# EPICS substitutions: blenApp/Db/common/IMAXScale.substitutions
#==============================================================================
#
# Abs:  IMAX scale substitutions file.
#
# Name: IMAXScale.substitutions
#
# Note: Must follow the LCLS naming conventions.
#
#==============================================================================
#
file IMAXScaleCalc.db
{
pattern   {P, SCAN}

# P is the PV prefix
# SCAN is the SCAN field

          { $(P), "1 second"}
}
